ABB RobotStudio station: RA projekat ABB.rspag

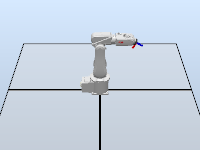
--- station ---
Station RA projekat ABB (saved by RobotStudio 21.1.9393.1)
Controller IRB120_3_58
  mechanical unit ROB_1: IRB120_3_58__01, 6 joints, base frame (0, 0, 0) mm
Layout (positions relative to the parent item):
  - IRB120_3_58__01 [mechanism, from Robots\IRB120_3_58_G_01.rslib] at (0, 0, 0) mm; joint values [0, 0, 0, 0, 0.5236, 0] (rad or m)

--- Backups/IRB120_3_58/RAPID/TASK1/PROGMOD/Module1.mod ---
MODULE Module1
    !***********************************************************
    !
    ! Module:  Module1
    !
    ! Description:
    !   <Insert description here>
    !
    ! Author: Marija
    !
    ! Version: 1.0
    !
    !***********************************************************


    !***********************************************************
    !
    ! Procedure main
    !
    !   This is the entry point of your program
    !
    !***********************************************************

    VAR num callCount;

!Get a random number between 0 and 1
FUNC NUM CheckWeld()
VAR num val:=1;


var pos pos_current;
pos_current := CPos(\Tool:=tool0 \WObj:=wobj0);

!1 seeding, Seed by position
val:=val*(Abs(ROUND(pos_current.x*100, \Dec:=0)) +1); !+1 to avoid mul by 0 scenario
val := 789 + val MOD 1000; !777 is just a bogus valu, since the mod might give 0

!Feel free to seed with y,z, more

!2. seeding, Seed by time
val :=val * ( GetTime(\Sec)+1);
val :=val * ( GetTime(\Min)+1);


!3 seeding, increment callcount and handle large number
callCount := callCount +1;
IF callCount > 1000 THEN
    callCount := 234;
ENDIF

!finally a division to get something interesting large float number
val := val / callCount;

!get a value between 0 and 1 using COS ( math)
RETURN (0.5 + COS(val)/2)*100;

ENDFUNC

    PROC main()
        !Add your code here
    ENDPROC
ENDMODULE

--- Backups/IRB120_3_58/SYSPAR/EIO.cfg ---
EIO:CFG_1.0:6:1::
#
EIO_SIGNAL:

      -Name "WeldinGun" -SignalType "DO"

      -Name "WledingPass" -SignalType "DO"

      -Name "WeldingFail" -SignalType "DO"
